FUNCTION_BLOCK TcoMessengerContextTest EXTENDS TcoCore._internals_TcoContext
VAR
	_CallMyPlcInstance 		:	BOOL := FALSE;
	_TcoMessangerTests		:	TcoMessengerTests(THIS^);
	_RtcIsValid				:	BOOL;
END_VAR

IF THIS^._CallMyPlcInstance THEN
	THIS^.Run();
	THIS^.RtcIsValid();
END_IF

{attribute 'TcRpcEnable'}
METHOD INTERNAL ContextClose
SUPER^._Close();
END_METHOD

{attribute 'TcRpcEnable'}
METHOD INTERNAL ContextOpen
SUPER^._Open();
END_METHOD

METHOD PROTECTED  Main
END_METHOD

{attribute 'TcRpcEnable'}
METHOD INTERNAL RtcIsValid : BOOL
RtcIsValid := THIS^.Rtc.IsValid;
_RtcIsValid := THIS^.Rtc.IsValid;
END_METHOD

END_FUNCTION_BLOCK

(* stored: Version 1.1.0.1, ProductVersion 3.1.4024.6
   POU TcoMessengerContextTest: Id {ab1f1c15-693e-0b9d-1dc8-8f3fbcb09dcf}, SpecialFunc None
   Method ContextClose: Id {4f2fdfc4-fcab-0528-13d7-8604dcba8327}
   Method ContextOpen: Id {89a806dd-7d63-036b-0493-cf31446222af}
   Method Main: Id {ce1913c5-df6b-0aa3-3f90-ae6b899c0533}
   Method RtcIsValid: Id {26119aec-f827-0ffc-3e54-5571e4e4da19} *)
